// Mitsubishi GX Works2 project: 오목_프로젝트완   PLC: Q03UDV

PROGRAM MAIN
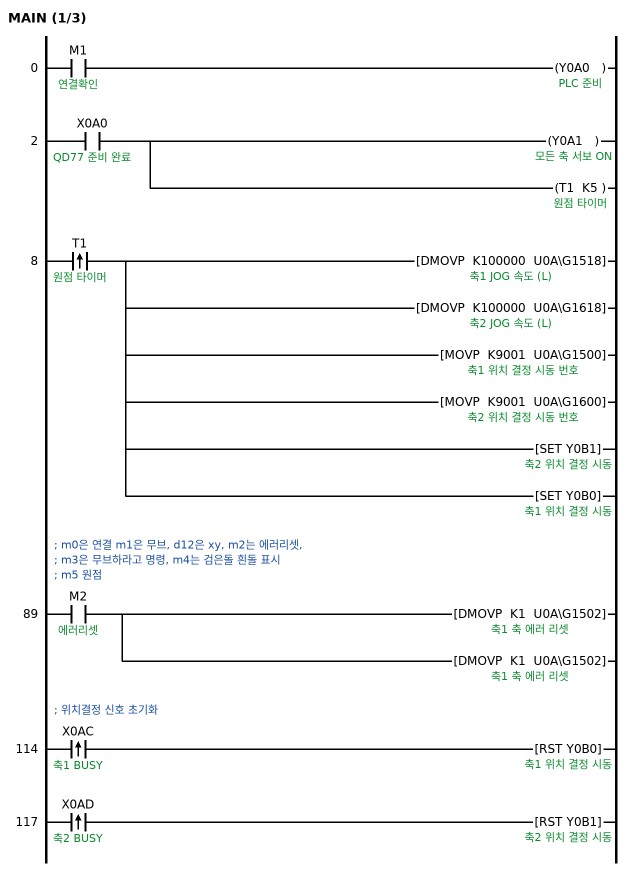
0     LD      M1  ; 연결확인
      OUT     Y0A0  ; PLC 준비
2     LD      X0A0  ; QD77 준비 완료
      OUT     Y0A1  ; 모든 축 서보 ON
      OUT     T1 K5  ; 원점 타이머
8     LDP     T1  ; 원점 타이머
      DMOVP   K100000 U0A\G1518  ; 축1 JOG 속도 (L)
      DMOVP   K100000 U0A\G1618  ; 축2 JOG 속도 (L)
      MOVP    K9001 U0A\G1500  ; 축1 위치 결정 시동 번호
      MOVP    K9001 U0A\G1600  ; 축2 위치 결정 시동 번호
      SET     Y0B1  ; 축2 위치 결정 시동
      SET     Y0B0  ; 축1 위치 결정 시동
; m0은 연결 m1은 무브, d12은 xy, m2는 에러리셋,
; m3은 무브하라고 명령, m4는 검은돌 흰돌 표시
; m5 원점
89    LD      M2  ; 에러리셋
      DMOVP   K1 U0A\G1502  ; 축1 축 에러 리셋
      DMOVP   K1 U0A\G1502
; 위치결정 신호 초기화
114   LDP     X0AC  ; 축1 BUSY
      RST     Y0B0  ; 축1 위치 결정 시동
117   LDP     X0AD  ; 축2 BUSY
      RST     Y0B1  ; 축2 위치 결정 시동
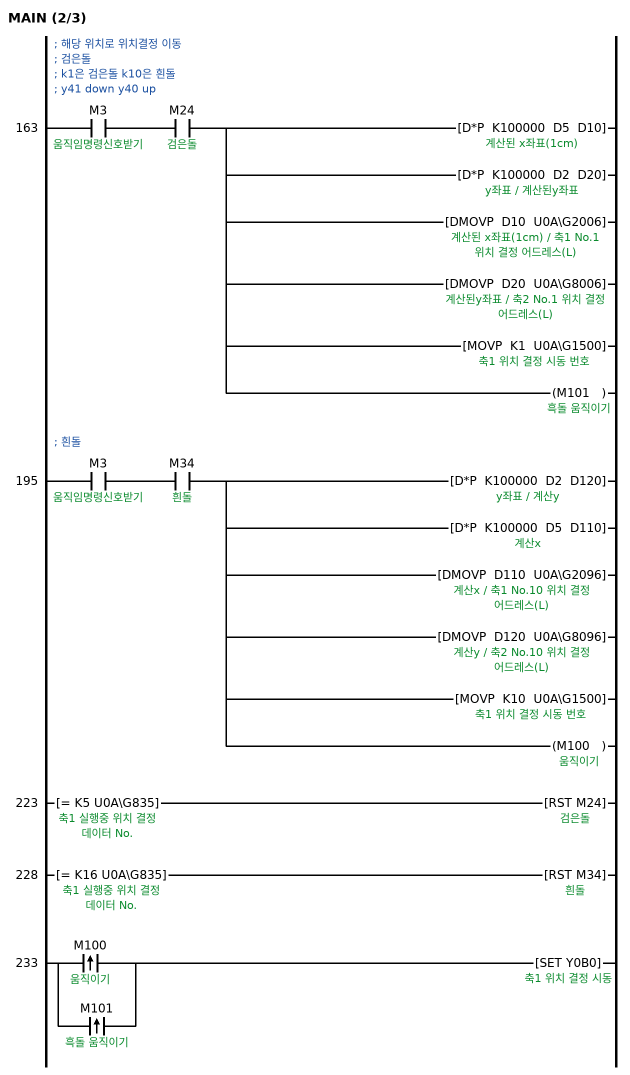
; 해당 위치로 위치결정 이동
; 검은돌
; k1은 검은돌 k10은 흰돌
; y41 down y40 up
163   LD      M3  ; 움직임명령신호받기
      AND     M24  ; 검은돌
      D*P     K100000 D5 D10  ; 계산된 x좌표(1cm)
      D*P     K100000 D2 D20  ; y좌표 / 계산된y좌표
      DMOVP   D10 U0A\G2006  ; 축1 No.1 위치 결정 어드레스(L)
      DMOVP   D20 U0A\G8006  ; 축2 No.1 위치 결정 어드레스(L)
      MOVP    K1 U0A\G1500
      OUT     M101  ; 흑돌 움직이기
; 흰돌
195   LD      M3  ; 움직임명령신호받기
      AND     M34  ; 흰돌
      D*P     K100000 D2 D120  ; 계산y
      D*P     K100000 D5 D110  ; 계산x
      DMOVP   D110 U0A\G2096  ; 축1 No.10 위치 결정 어드레스(L)
      DMOVP   D120 U0A\G8096  ; 축2 No.10 위치 결정 어드레스(L)
      MOVP    K10 U0A\G1500
      OUT     M100  ; 움직이기
223   LD=     K5 U0A\G835  ; 축1 실행중 위치 결정 데이터 No.
      RST     M24  ; 검은돌
228   LD=     K16 U0A\G835  ; 축1 실행중 위치 결정 데이터 No.
      RST     M34  ; 흰돌
233   LDP     M100  ; 움직이기
      ORP     M101  ; 흑돌 움직이기
      SET     Y0B0  ; 축1 위치 결정 시동
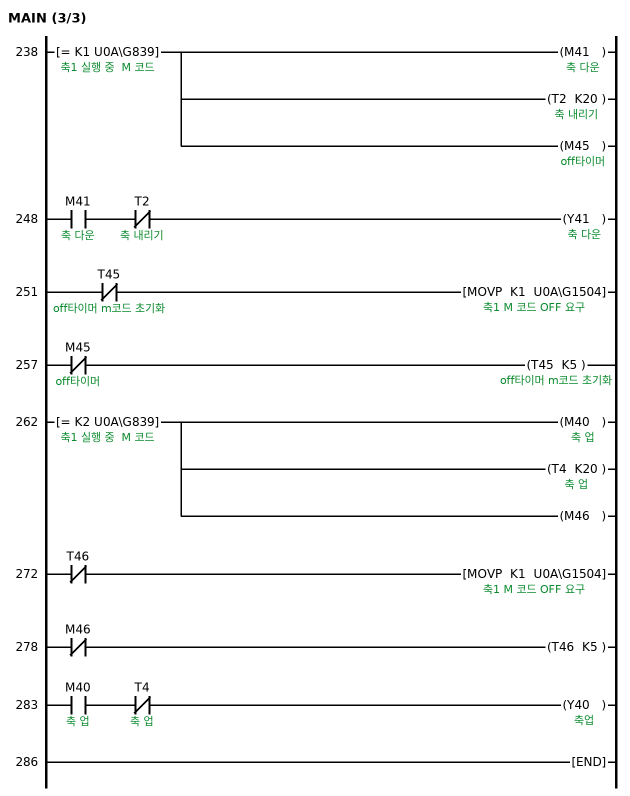
238   LD=     K1 U0A\G839  ; 축1 실행 중  M 코드
      OUT     M41  ; 축 다운
      OUT     T2 K20  ; 축 내리기
      OUT     M45  ; off타이머
248   LD      M41  ; 축 다운
      ANI     T2  ; 축 내리기
      OUT     Y41  ; 축 다운
251   LDI     T45  ; off타이머 m코드 초기화
      MOVP    K1 U0A\G1504  ; 축1 M 코드 OFF 요구
257   LDI     M45  ; off타이머
      OUT     T45 K5  ; off타이머 m코드 초기화
262   LD=     K2 U0A\G839  ; 축1 실행 중  M 코드
      OUT     M40  ; 축 업
      OUT     T4 K20  ; 축 업
      OUT     M46
272   LDI     T46
      MOVP    K1 U0A\G1504
278   LDI     M46
      OUT     T46 K5
283   LD      M40  ; 축 업
      ANI     T4  ; 축 업
      OUT     Y40  ; 축업
286   END
END_PROGRAM

// device comments not shown above
X0A1  ; 동기용 플래그
X0A4  ; 축1 M 코드 ON
X0A5  ; 축2 M 코드 ON
X0A8  ; 축1 에러 검출
X0A9  ; 축2 에러 검출
X0B0  ; 축1 시동 완료
X0B1  ; 축2 시동 완료
X0B4  ; 축1 위치 결정 완료
X0B5  ; 축2 위치 결정 완료
Y0A4  ; 축1 축 정지
Y0A5  ; 축2 축 정지
Y0A8  ; 축1 정운전 JOG 시동
Y0A9  ; 축1 역운전 JOG 시동
Y0AA  ; 축2 정운전 JOG 시동
Y0AB  ; 축2 역운전 JOG 시동
Y0B4  ; 축1 실행 금지 플래그
Y0B5  ; 축2 실행 금지 플래그
D0  ; x좌표
M4  ; f검은돌t흰돌
M5  ; 원점
M33  ; 리셋신호
M50  ; 무브 신호
M102  ; 원점 움직이기
T3  ; 원점 종료
T20  ; m코드 초기화
T40  ; m코드 초기화
